TYPE ST_AXIS_LIMIT_SWITCHES :
STRUCT
  bMinimum      : BOOL;
  bMaximum      : BOOL;
  bCalibrate    : Bool;
END_STRUCT
END_TYPE

(* stored: Version 1.1.0.1, ProductVersion 3.1.4026.13
   DUT ST_AXIS_LIMIT_SWITCHES: Id {8ff35ecf-1770-448d-b3f0-a063a0cf77f1} *)
